      MachineInterface.MotionsStandStill := Sts.IsStandstill;

      MachineInterface.AutReady := AreaInterface.Aut AND NOT Sts.AlarmsPresence;


      MachineInterface.AckStopInPhase := AreaInterface.StopInPhase AND Ctrl.Stop;

      MachineInterface.AckStopProgrammed := AreaInterface.StopProgrammed AND Ctrl.Stop;


      MachineInterface.Aborting := AreaInterface.Aut AND Sts.AlarmsPresence;


   END_REGION


END_FUNCTION_BLOCK
